// TIA Portal V16 export
// export: Created 2024-12-03T15:41:45.2667557Z, ExportSetting WithReadOnly, DisplayName Totally Integrated Automation Portal, DisplayVersion V16 Update 6, DisplayName TIA Portal Version Control Interface, DisplayVersion V16 Update 2, DisplayName TIA Portal Openness, DisplayVersion V16 Update 6, DisplayName TIA Portal Teamcenter Gateway, DisplayVersion V16, DisplayName SINAMICS Startdrive Advanced, DisplayVersion V16 Update 5, DisplayName SINAMICS Startdrive G130, G150, S120, S150, SINAMICS MV, S210, DisplayVersion V16 Update 5, DisplayName SINAMICS Startdrive G110M, G120, G120C, G120D, G120P, G115D, DisplayVersion V16 Update 5, DisplayName STEP 7 Professional, DisplayVersion V16 Update 6, DisplayName STEP 7 Safety, DisplayVersion V16, DisplayName WinCC Advanced / Unified PC, DisplayVersion V16 Update 6
TYPE "COGNEX_DATAMAN_IN_UDT"
// stored: CreationDate 2022-02-10T08:20:21.8932261Z, InterfaceModifiedDate 2020-06-23T05:35:36.0351598Z, IsConsistent true, LibraryConformanceStatus The object is library-conformant., ModifiedDate 2020-06-23T22:30:53.6218309Z
   STRUCT
      Status_TriggerReady : Bool;   // 0 = Not Ready to Accept Trigger via Fieldbus (statewhen Trigger Enable is low or currently processingtrigger or soft event)1 = Ready to Accept new Trigger via Fieldbus
      Status_TriggerAck : Bool;   // Confirmation of receiving Trigger ON bit, stays on untilTrigger bit is low
      Status_Acquiring : Bool;   // 0 = Reader Idle1 = Reader Processing a trigger (whether it came fromphoto eye or fieldbus)
      Status_MissedTrigger : Bool;   // 0 = No Error1 = Received a trigger (signal from Photo Eye or Fieldbus) when an other trigger or soft event is processing.Will reset automatically when a successful trigger couldbe processed again.
      Status_CurrentMode : Bool;   // 0 = Setup Tool Mode1 = Run Mode
      Status_SerialError : Bool;   // 0 = No Error; Reader is Connected1 = No Reader connected
      Status_TrigerPin4State : Bool;   // Copy state of input line IN 1
      Status_TriggerPin2State : Bool;   // Copy state of input line IN 2
      ResultStatus_ResultAvailable : Bool;   // Indicates that a new set of read results are available (i.e.the contents of the Result Data are valid). Cleared whenresults are acknowledged by PLC
      ResultStatus_ResultAckMirror : Bool;   // This bit mirrors the state of the "Results Ack" bit from theoutput data. This is not exactly "Result Data Valid".When the result data is first presented, this bit will still be"0," since it just mirrors the "Results Ack" bit from the lastoutput but the data is valid.
      ResultStatus_ResultDataBufferOverFlow : Bool;
      ResultStatus_spare_1 : Bool;
      ResultStatus_spare_2 : Bool;
      ResultStatus_spare_3 : Bool;
      ResultStatus_spare_4 : Bool;
      ResultStatus_GeneralFault : Bool;
      SoftEventStatus_errorCode1 : Bool;   // Soft event error code from DMCCError code 127 - timeout
      SoftEventStatus_errorCode2 : Bool;
      SoftEventStatus_errorCode3 : Bool;
      SoftEventStatus_errorCode4 : Bool;
      SoftEventStatus_errorCode5 : Bool;
      SoftEventStatus_errorCode6 : Bool;
      SoftEventStatus_errorCode7 : Bool;
      SoftEventStatus_CommendTimedOutOrCompleted : Bool;
      ResultCode_TriggerResult : Bool;
      ResultCode_SoftCommandIsRunning : Bool;
      ResultCode_SoftCommandComplete : Bool;
      ResultCode_spare_3 : Bool;
      ResultCode_spare_4 : Bool;
      ResultCode_spare_5 : Bool;
      ResultCode_spare_6 : Bool;
      ResultCode_spare_7 : Bool;
      TriggerId : Byte;   // ID value of the next trigger to be issued. Used to matchissues triggers with corresponding result data receivedlater.
      ResultId : Byte;   // The value of the “Trigger ID” counter when the triggerthat generated these results was issued.
      ResultLength : Byte;   // Actual number of bytes contained in the “Result Data"field
      DataBlock_DataBlockSize_0 : Bool;
      DataBlock_DataBlockSize_1 : Bool;
      DataBlock_DataBlockSize_2 : Bool;
      DataBlock_DataBlockSize_3 : Bool;
      DataBlock_spare_4 : Bool;
      DataBlock_spare_5 : Bool;
      DataBlock_spare_6 : Bool;
      DataBlock_Reader2Disabled : Bool;   // 0 = Reader 2 Enabled (default)1 = Reader 2 Disabled
      Barcode : Array[0..135] of Char;
   END_STRUCT;
END_TYPE
